SYSTEM Kulbana System
  (* Version 1.0, 2005-06-13, Goran, Chalmers *)
  DEVICE Test Device : DeviceType_not_used
    RESOURCE TestResource : ResourceType_not_used
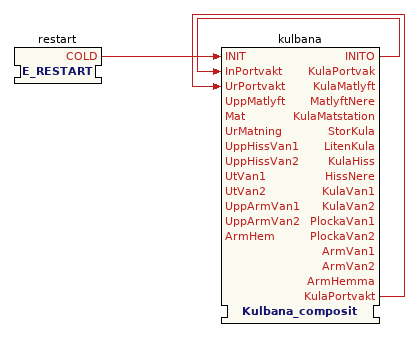
      FBS
        restart : E_RESTART;
        kulbana : Kulbana_composit;
      END_FBS
      EVENT_CONNECTIONS
        restart.COLD TO kulbana.INIT;
        kulbana.INITO TO kulbana.InPortvakt;
        kulbana.KulaPortvakt TO kulbana.UrPortvakt;
      END_CONNECTIONS
    END_RESOURCE
  END_DEVICE
END_SYSTEM
